FUNCTION_BLOCK MasterSlave_TEST (* Composite Function Block Type *)
  (* Standard: 61499-2 *)
  (* Version 0.0, 2011-03-19, Majid Sorouri, nxtControl GmbH, template *)
  (* Compiler header: package fb.rt.pnp; *)
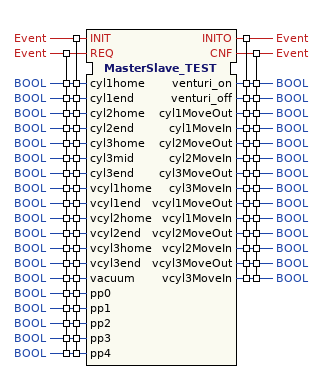
  EVENT_INPUT
    INIT WITH vacuum, pp0, pp1, pp2, pp3, cyl1home, cyl1end, cyl2home, cyl2end, cyl3home, cyl3mid, cyl3end, vcyl1home, vcyl1end, vcyl2home, vcyl2end, vcyl3home, vcyl3end, pp4; (* Initialization Request *)
    REQ WITH vacuum, pp0, pp1, pp2, pp3, cyl1home, cyl1end, cyl2home, cyl2end, cyl3home, cyl3mid, cyl3end, vcyl1home, vcyl1end, vcyl2home, vcyl2end, vcyl3home, vcyl3end, pp4; (* Normal Execution Request *)
  END_EVENT
  EVENT_OUTPUT
    INITO WITH venturi_off, venturi_on, cyl1MoveOut, cyl1MoveIn, cyl2MoveOut, cyl2MoveIn, cyl3MoveOut, cyl3MoveIn, vcyl1MoveOut, vcyl1MoveIn, vcyl2MoveOut, vcyl2MoveIn, vcyl3MoveOut, vcyl3MoveIn; (* Initialization Confirm *)
    CNF WITH venturi_on, venturi_off, cyl1MoveOut, cyl1MoveIn, cyl2MoveOut, cyl2MoveIn, cyl3MoveOut, cyl3MoveIn, vcyl1MoveOut, vcyl1MoveIn, vcyl2MoveOut, vcyl2MoveIn, vcyl3MoveOut, vcyl3MoveIn; (* Execution Confirmation *)
  END_EVENT
  VAR_INPUT
    cyl1home : BOOL;
    cyl1end : BOOL;
    cyl2home : BOOL;
    cyl2end : BOOL;
    cyl3home : BOOL;
    cyl3mid : BOOL;
    cyl3end : BOOL;
    vcyl1home : BOOL;
    vcyl1end : BOOL;
    vcyl2home : BOOL;
    vcyl2end : BOOL;
    vcyl3home : BOOL;
    vcyl3end : BOOL;
    vacuum : BOOL;
    pp0 : BOOL;
    pp1 : BOOL;
    pp2 : BOOL;
    pp3 : BOOL;
    pp4 : BOOL;
  END_VAR
  VAR_OUTPUT
    venturi_on : BOOL;
    venturi_off : BOOL;
    cyl1MoveOut : BOOL;
    cyl1MoveIn : BOOL;
    cyl2MoveOut : BOOL;
    cyl2MoveIn : BOOL;
    cyl3MoveOut : BOOL;
    cyl3MoveIn : BOOL;
    vcyl1MoveOut : BOOL;
    vcyl1MoveIn : BOOL;
    vcyl2MoveOut : BOOL;
    vcyl2MoveIn : BOOL;
    vcyl3MoveOut : BOOL;
    vcyl3MoveIn : BOOL;
  END_VAR
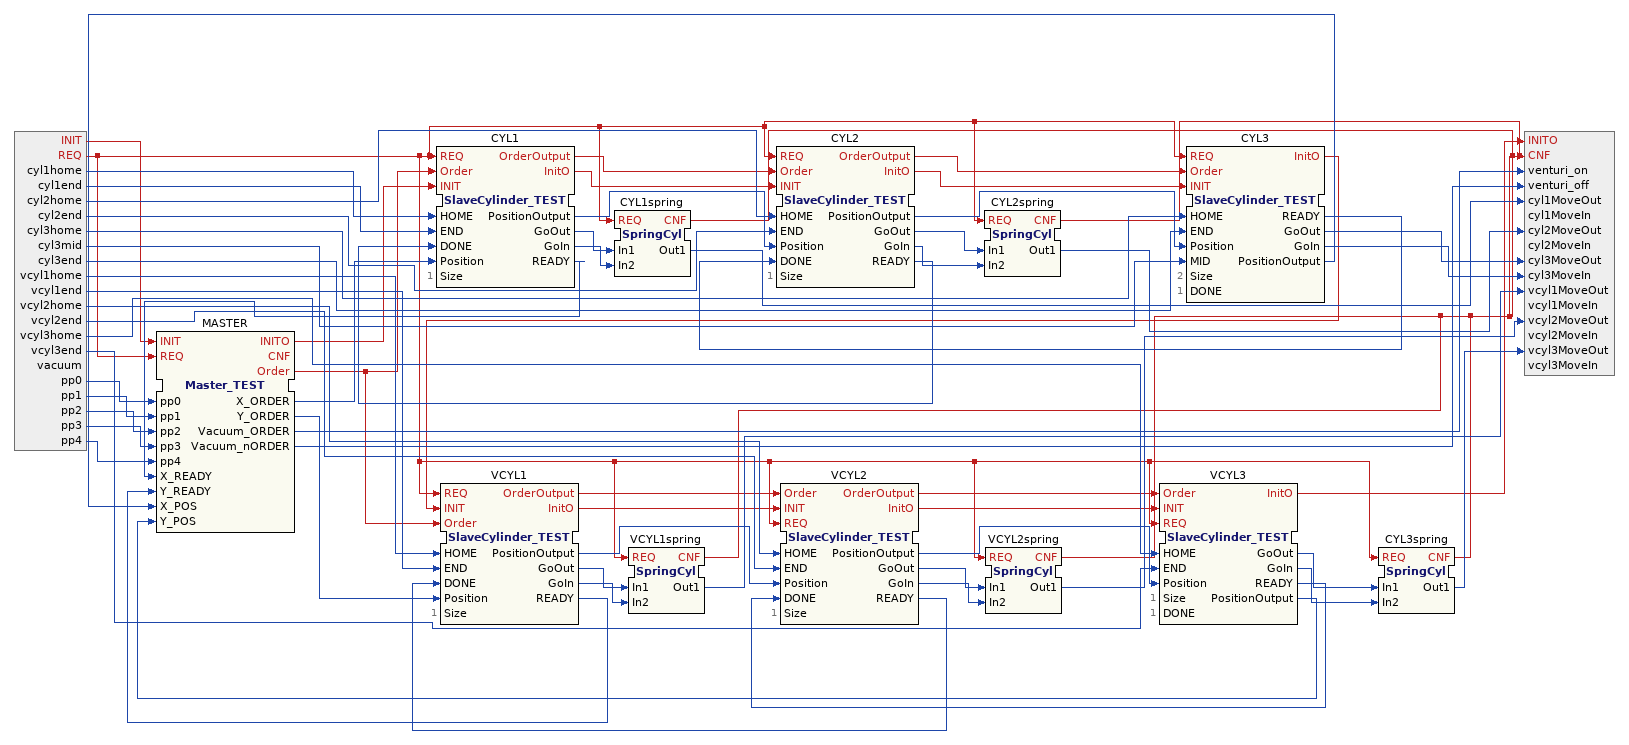
  FBS
    CYL3spring : SpringCyl;
    CYL1spring : SpringCyl;
    VCYL1spring : SpringCyl;
    CYL2spring : SpringCyl;
    VCYL2spring : SpringCyl;
    CYL1 : SlaveCylinder_TEST(Size := 1);
    CYL2 : SlaveCylinder_TEST(Size := 1);
    CYL3 : SlaveCylinder_TEST(Size := 2, DONE := 1);
    VCYL1 : SlaveCylinder_TEST(Size := 1);
    VCYL2 : SlaveCylinder_TEST(Size := 1);
    VCYL3 : SlaveCylinder_TEST(Size := 1, DONE := 1);
    MASTER : Master_TEST;
  END_FBS
  EVENT_CONNECTIONS
    CYL1spring.CNF TO CNF;
    VCYL1spring.CNF TO CNF;
    VCYL2spring.CNF TO CNF;
    CYL2spring.CNF TO CNF;
    REQ TO CYL2spring.REQ;
    REQ TO VCYL2spring.REQ;
    CYL3spring.CNF TO CNF;
    REQ TO CYL3spring.REQ;
    REQ TO CYL3.REQ;
    REQ TO CYL2.REQ;
    REQ TO CYL1.REQ;
    CYL1.OrderOutput TO CYL2.Order;
    CYL2.OrderOutput TO CYL3.Order;
    CYL2.InitO TO CYL3.INIT;
    CYL1.InitO TO CYL2.INIT;
    VCYL1.OrderOutput TO VCYL2.Order;
    VCYL2.OrderOutput TO VCYL3.Order;
    VCYL2.InitO TO VCYL3.INIT;
    VCYL1.InitO TO VCYL2.INIT;
    REQ TO VCYL2.REQ;
    REQ TO VCYL3.REQ;
    REQ TO VCYL1.REQ;
    REQ TO VCYL1spring.REQ;
    REQ TO CYL1spring.REQ;
    CYL3.InitO TO VCYL1.INIT;
    MASTER.Order TO CYL1.Order;
    MASTER.Order TO VCYL1.Order;
    INIT TO MASTER.INIT;
    REQ TO MASTER.REQ;
    MASTER.INITO TO CYL1.INIT;
    VCYL3.InitO TO INITO;
  END_CONNECTIONS
  DATA_CONNECTIONS
    CYL1spring.Out1 TO cyl1MoveOut;
    VCYL1spring.Out1 TO vcyl1MoveOut;
    CYL2spring.Out1 TO cyl2MoveOut;
    VCYL2spring.Out1 TO vcyl2MoveOut;
    CYL3spring.Out1 TO vcyl3MoveOut;
    cyl1home TO CYL1.HOME;
    cyl1end TO CYL1.END;
    cyl2home TO CYL2.HOME;
    cyl2end TO CYL2.END;
    cyl3home TO CYL3.HOME;
    cyl3end TO CYL3.END;
    vcyl1home TO VCYL1.HOME;
    vcyl1end TO VCYL1.END;
    vcyl2home TO VCYL2.HOME;
    vcyl2end TO VCYL2.END;
    vcyl3home TO VCYL3.HOME;
    vcyl3end TO VCYL3.END;
    CYL1.PositionOutput TO CYL2.Position;
    CYL2.PositionOutput TO CYL3.Position;
    VCYL1.PositionOutput TO VCYL2.Position;
    VCYL2.PositionOutput TO VCYL3.Position;
    CYL1.GoOut TO CYL1spring.In1;
    CYL1.GoIn TO CYL1spring.In2;
    CYL2.GoOut TO CYL2spring.In1;
    CYL2.GoIn TO CYL2spring.In2;
    VCYL1.GoOut TO VCYL1spring.In1;
    VCYL1.GoIn TO VCYL1spring.In2;
    VCYL2.GoOut TO VCYL2spring.In1;
    VCYL2.GoIn TO VCYL2spring.In2;
    VCYL3.GoOut TO CYL3spring.In1;
    VCYL3.GoIn TO CYL3spring.In2;
    CYL2.READY TO CYL1.DONE;
    CYL3.READY TO CYL2.DONE;
    VCYL3.READY TO VCYL2.DONE;
    VCYL2.READY TO VCYL1.DONE;
    CYL3.GoOut TO cyl3MoveOut;
    CYL3.GoIn TO cyl3MoveIn;
    MASTER.X_ORDER TO CYL1.Position;
    MASTER.Y_ORDER TO VCYL1.Position;
    VCYL3.PositionOutput TO MASTER.Y_POS;
    CYL3.PositionOutput TO MASTER.X_POS;
    VCYL1.READY TO MASTER.Y_READY;
    CYL1.READY TO MASTER.X_READY;
    pp0 TO MASTER.pp0;
    pp1 TO MASTER.pp1;
    pp2 TO MASTER.pp2;
    pp3 TO MASTER.pp3;
    pp4 TO MASTER.pp4;
    MASTER.Vacuum_ORDER TO venturi_on;
    MASTER.Vacuum_nORDER TO venturi_off;
    cyl3mid TO CYL3.MID;
  END_CONNECTIONS
END_FUNCTION_BLOCK
